// TIA Portal project "Sensor_Valve_Activate" (V16)

(* hardware
DEVICE "S7-1200 station_1"  S7-1200 Station
   slot 0: "Rack_0"  S7-1200 Rack  Rack  V1.0
   slot 1: "PLC_1"  CPU 1214C DC/DC/DC  6ES7 214-1AG40-0XB0  V4.2
*)

// ===== PLC "PLC_1"  CPU 1214C DC/DC/DC =====

VAR_GLOBAL   // PLC tag table "Default tag table"
   ""i_xSupply_InletValve_Open_A1"" AT %I0.1 : Bool;
   ""i_xSupply_FeedPump_Running_A1"" AT %I2.1 : Bool;
   ""i_xSupply_FeedValve_Open_A1"" AT %I0.0 : Bool;
   ""i_xSupply_FlowSensor_A1"" AT %I0.5 : Bool;
   ""i_xMix_Motor_Running"" AT %I4.1 : Bool;
   ""i_xDrain_SolenoidValve_Open"" AT %I2.5 : Bool;
   ""i_xButtonFeedPump_Start_A1"" AT %I30.3 : Bool;
   ""i_xButtonFeedPump_Stop_A1"" AT %I30.4 : Bool;
   ""i_xButtonMotor_Start"" AT %I30.0 : Bool;
   ""i_xButtonMotor_Stop"" AT %I30.1 : Bool;
   ""i_xButtonSolenoidValve_Start"" AT %I31.0 : Bool;
   ""i_xButtonSolenoidValve_Stop"" AT %I31.1 : Bool;
   ""i_xButtonMaintenanceLamp_Stop"" AT %I10.6 : Bool;
   ""i_xButton_Emergency"" AT %I10.7 : Bool;
   ""i_xSupply_InletValve_Open_A2"" AT %I0.3 : Bool;
   ""i_xSupply_FeedPump_Running_A2"" AT %I2.7 : Bool;
   ""i_xSupply_FeedValve_Open_A2"" AT %I0.2 : Bool;
   ""i_xSupply_FlowSensor_A2"" AT %I0.6 : Bool;
   ""i_xMix_Tank_EmptySensor"" AT %I0.4 : Bool;
   ""i_xButtonFeedPump_Start_A2"" AT %I30.5 : Bool;
   ""i_xButtonFeedPump_Stop_A2"" AT %I30.6 : Bool;
   ""i_xSupply_FeedPump_Ready_A1"" AT %I3.5 : Bool;
   ""i_xSupply_FeedPump_Ready_A2"" AT %I3.6 : Bool;
   ""i_xDrain_SolenoidValve_Close"" AT %I2.3 : Bool;
   ""i_xButton_Reset"" AT %I30.2 : Bool;
   ""i_xMix_Motor_Stop"" AT %I4.0 : Bool;
   ""i_xButton_Turn/off_Maintenance_Pump"" AT %I31.3 : Bool;
   ""i_xButton_Turn/off_Maintenance_Motor"" AT %I31.2 : Bool;
   ""iq_xMix_Tank_FullSensor"" AT %I7.7 : Bool;
   ""i_xFull_Sensor"" AT %I8.0 : Bool;
   ""q_xSupply_FeedPump_Start_A1"" AT %Q3.0 : Bool;
   ""q_xSupply_InletValve_Open_A1"" AT %Q3.2 : Bool;
   ""q_xLamp_Running"" AT %Q4.0 : Bool;
   ""q_xLamp_Faulted"" AT %Q4.1 : Bool;
   ""q_xMix_Motor_Start"" AT %Q6.4 : Bool;
   ""q_xDrain_SolenoidValve_Open"" AT %Q3.7 : Bool;
   ""q_xSupply_FeedPump_Start_A2"" AT %Q3.1 : Bool;
   ""q_xSupply_InletValve_Open_A2"" AT %Q3.3 : Bool;
   ""q_xSupply_FeedValve_Open_A1"" AT %Q3.4 : Bool;
   ""q_xSupply_FeedValve_Open_A2"" AT %Q3.5 : Bool;
   ""q_xLamp_Pump_Start_A1"" AT %Q4.2 : Bool;
   ""q_xLamp_Pump_Stop_A1"" AT %Q4.3 : Bool;
   ""q_xLamp_Pump_Start_A2"" AT %Q4.4 : Bool;
   ""q_xLamp_Pump_Stop_A2"" AT %Q4.5 : Bool;
   ""q_xLamp_Motor_Start"" AT %Q4.6 : Bool;
   ""q_xLampSolenoidValve_Start"" AT %Q5.0 : Bool;
   ""q_xLampSolenoidValve_Stop"" AT %Q5.1 : Bool;
   ""q_xLamp_Pump_Maintain_A1"" AT %Q5.2 : Bool;
   ""q_xLamp_Pump_Maintain_A2"" AT %Q5.3 : Bool;
   ""q_xLamp_Motor_Stop"" AT %Q4.7 : Bool;
   ""q_xLamp_Motor_Maintain"" AT %Q5.4 : Bool;
   ""q_xLamp_Tank_Full"" AT %Q5.5 : Bool;
   ""q_xLamp_Tank_Empty"" AT %Q5.6 : Bool;
   ""q_xLamp_Emergency"" AT %Q5.7 : Bool;
   ""q_xDisp_Tank_Level"" AT %QD60 : DWord;
   ""q_xDisp_Motor_Speed"" AT %QD64 : DWord;
   ""q_xSupply_FeedPump_Stop_A1"" AT %Q6.0 : Bool;
   ""q_xSupply_FeedPump_Stop_A2"" AT %Q6.1 : Bool;
   ""q_xDrain_SolenoidValve_Close"" AT %Q2.7 : Bool;
   ""q_xMix_Motor_Stop"" AT %Q6.5 : Bool;
   ""q_xMaintain_Lamp_Motor"" AT %Q10.1 : Bool;
   ""q_xMaintain_Lamp_Pump"" AT %Q10.2 : Bool;
   ""q_xLamp_Fault"" AT %Q120.1 : Bool;
END_VAR